// TwinCAT 3 PLC project Untitled1
// ProgramVersion: 3.1.4026.12
// libraries:
//   Tc2_Standard, * (Beckhoff Automation GmbH)
//   Tc2_System, * (Beckhoff Automation GmbH)
//   Tc3_Module, * (Beckhoff Automation GmbH)
// project tree:
//   / PlcTask.TcTTO
//   POUs/ FB_Calculation.TcPOU, MAIN.TcPOU
// (motion and I/O tree: see PLC project flc)
// real-time tasks:
//   TASK StateMachine: cycle T#5ms, priority 8, ADS port 350
//   TASK ModbusComm: cycle T#20ms, priority 12, ADS port 351
//   TASK TimerTask: cycle T#1ms, priority 6, ADS port 353
//   TASK EAPControl_Task: cycle T#800us, priority 4, ADS port 354
//   TASK PlcTask: cycle T#10ms, priority 10, ADS port 352
// variable links:

CONFIGURATION Untitled1
    RESOURCE PLC ON TwinCAT3
        TASK PlcTask(INTERVAL := T#10ms, PRIORITY := 10);
        PROGRAM MAIN WITH PlcTask : MAIN;
    END_RESOURCE
END_CONFIGURATION

// ---- POUs/MAIN.TcPOU
PROGRAM MAIN
VAR
END_VAR

END_PROGRAM

// ---- POUs/FB_Calculation.TcPOU
FUNCTION_BLOCK FB_Calculation EXTENDS TcBaseModuleRegistered
VAR_INPUT
END_VAR
VAR_OUTPUT
END_VAR
VAR
END_VAR

END_FUNCTION_BLOCK
